FUNCTION_BLOCK PUBLIC Stack_TestSuite EXTENDS TcUnit.FB_TestSuite

// check datatypes are handled correctly
CheckListWorksWithIntegers();
CheckListWorksWithStrings();
CheckListWorksWithArrays();

// all other checks
CheckStackImplementsI_Stack();
CheckContains();
CheckClear();
CheckCount();
CheckAddItem();
CheckTryRemoveItem();
CheckTryPopRemovesTheItem();
CheckTryPopReturnsTheCorrectValue();
CheckTryPeekReturnsTheCorrectValue();
CheckTryPeekDoesNotRemoveTheItem();
CheckOnChangedEvent();
CheckOnDisposedEvent();
CheckOnceEvent();
CheckOffEvent();
CheckTryCopyTo();
CheckTryCopyToLocation();
CheckStackOrderIsCorrect();
CheckListReturnsEnumerator();
CheckEnumeratorIsInvalidAfterChange();
CheckIsEmptyWhenEmpty();
CheckIsEmptyWhenFull();

METHOD PUBLIC CheckAddItem
VAR
	in1 : INT := 123;
	in2 : INT := 456;
	in3 : INT := 789;
	result : BOOL;
	stack : Stack;
END_VAR
TEST('CheckAddItem');

// @TEST-FIXTURE
stack.Push(in1); // (fifo->) 123
stack.Push(in2); // (fifo->) 456, 123

// @TEST-RUN
stack.AddItem(in3); // fifo->) 789, 456, 123
result := stack.Contains(in3);

// @TEST-ASSSERT
AssertTrue(
	Condition := result,
	Message := 'Method returned false'
);

TEST_FINISHED();
END_METHOD

METHOD PUBLIC CheckClear
VAR
	in1 : INT := 123;
	in2 : INT := 456;
	in3 : INT := 789;
	stack : Stack;
END_VAR
TEST('CheckClear');

// @TEST-FIXTURE
stack.Push(in1); // (fifo->) 123
stack.Push(in2); // (fifo->) 456, 123
stack.Push(in2); // (fifo->) 789, 456, 123

// @TEST-RUN
stack.Clear();

// @TEST-ASSSERT
AssertTrue(
	Condition := stack.Count = 0,
	Message := 'The count is not zero'
);

TEST_FINISHED();
END_METHOD

METHOD PUBLIC CheckContains
VAR
	in1 : INT := 123;
	in2 : INT := 456;
	in3 : INT := 789;
	result : BOOL;
	stack : Stack;
END_VAR
TEST('CheckContains');

// @TEST-FIXTURE
stack.Push(in1); // (fifo->) 123
stack.Push(in2); // (fifo->) 456, 123
stack.Push(in2); // (fifo->) 789, 456, 123

// @TEST-RUN
result := stack.Contains(in2);

// @TEST-ASSSERT
AssertTrue(
	Condition := result,
	Message := 'Did not find the item in the queue'
);

TEST_FINISHED();
END_METHOD

METHOD PUBLIC CheckCount
VAR
	in1 : INT := 123;
	in2 : INT := 456;
	in3 : INT := 789;
	total : DINT;
	expected : DINT := 3;
	stack : Stack;
END_VAR
TEST('CheckCount');

// @TEST-FIXTURE
stack.Push(in1); // (fifo->) 123
stack.Push(in2); // (fifo->) 456, 123
stack.Push(in2); // (fifo->) 789, 456, 123

// @TEST-RUN
total := stack.Count;

// @TEST-ASSSERT
AssertEquals(
	Expected := expected,
	Actual := total,
	Message := 'Incorrect count'
);

TEST_FINISHED();
END_METHOD

METHOD PUBLIC CheckEnumeratorIsInvalidAfterChange
VAR
	in : INT := 123;
	result : BOOL;
	stack : Stack;
	enumerator : I_ForwardEnumerator;
END_VAR
TEST('CheckEnumeratorIsInvalidAfterChange');

// @TEST-FIXTURE
enumerator := stack.GetEnumerator();
stack.Push(in);

// @TEST-RUN
result := enumerator.IsValid;
enumerator.Dispose();

// @TEST-ASSSERT
AssertFalse(
	Condition := result,
	Message := 'Method returned true'
);

TEST_FINISHED();
END_METHOD

METHOD PUBLIC CheckIsEmptyWhenEmpty
VAR
	result : BOOL;
	stack : Stack;
END_VAR
TEST('CheckIsEmptyWhenEmpty');

// @TEST-RUN
result := stack.IsEmpty;

// @TEST-ASSSERT
AssertTrue(
	Condition := result,
	Message := 'Incorrect state of IsEmpty'
);

TEST_FINISHED();
END_METHOD

METHOD PUBLIC CheckIsEmptyWhenFull
VAR
	in : INT := 123;
	result : BOOL;
	stack : Stack;
END_VAR
TEST('CheckIsEmptyWhenFull');

// @TEST-FIXTURE
stack.Push(in);

// @TEST-RUN
result := stack.IsEmpty;

// @TEST-ASSSERT
AssertFalse(
	Condition := result,
	Message := 'Incorrect state of IsEmpty'
);

TEST_FINISHED();
END_METHOD

METHOD PUBLIC CheckListReturnsEnumerator
VAR
	in1 : INT := 123;
	in2 : INT := 456;
	in3 : INT := 789;
	enumerator : I_ForwardEnumerator;
	stack : Stack;
END_VAR
TEST('CheckListReturnsEnumerator');

// @TEST-FIXTURE
stack.Push(in1); // (fifo->) 123
stack.Push(in2); // (fifo->) 456, 123
stack.Push(in2); // (fifo->) 789, 456, 123

// @TEST-RUN
enumerator := stack.GetEnumerator();

// @TEST-ASSSERT
AssertTrue(
	Condition := (enumerator <> 0),
	Message := 'Did not return an enumerator'
);

// @TEST-DISPOSE
enumerator.Dispose();

TEST_FINISHED();
END_METHOD

METHOD PUBLIC CheckListWorksWithArrays
VAR
	in : ARRAY [0..1] OF REAL := [0.1,2.3];
	out : ARRAY [0..1] OF REAL;
	expected : ARRAY [0..1] OF REAL := [0.1,2.3];
	result : BOOL;
	stack : Stack;
END_VAR
TEST('CheckListWorksWithArrays');

// @TEST-FIXTURE
stack.Push(in);

// @TEST-RUN
result := stack.TryPop(out);

// @TEST-ASSSERT
AssertTrue(
	Condition := result,
	Message := 'Method returned false'
);

AssertEquals(
	Expected := expected,
	Actual := out,
	Message := 'Did not produce the expected result'
);

TEST_FINISHED();
END_METHOD

METHOD PUBLIC CheckListWorksWithIntegers
VAR
	in : INT := 123;
	out : INT;
	expected : INT := 123;
	result : BOOL;
	stack : Stack;
END_VAR
TEST('CheckListWorksWithIntegers');

// @TEST-FIXTURE
stack.Push(in);

// @TEST-RUN
result := stack.TryPop(out);

// @TEST-ASSSERT
AssertTrue(
	Condition := result,
	Message := 'Method returned false'
);

AssertEquals(
	Expected := expected,
	Actual := out,
	Message := 'Did not produce the expected result'
);

TEST_FINISHED();
END_METHOD

METHOD PUBLIC CheckListWorksWithStrings
VAR
	in : STRING := 'test';
	out : STRING;
	expected : STRING := 'test';
	result : BOOL;
	stack : Stack;
END_VAR
TEST('CheckListWorksWithStrings');

// @TEST-FIXTURE
stack.Push(in);

// @TEST-RUN
result := stack.TryPop(out);

// @TEST-ASSSERT
AssertTrue(
	Condition := result,
	Message := 'Method returned false'
);

AssertEquals(
	Expected := expected,
	Actual := out,
	Message := 'Did not produce the expected result'
);

TEST_FINISHED();
END_METHOD

METHOD PUBLIC CheckOffEvent
VAR
	value : INT := 123;
	stack : Stack;
	handler : CollectionChangedEventHandler(ExpectedOriginator := stack);
END_VAR
TEST('CheckOffEvent');

// @TEST-FIXTURE
stack.OnEvent('OnChanged',handler);
stack.OffEvent('OnChanged',handler);

// @TEST-RUN
stack.Push(value);

// @TEST-ASSSERT
AssertFalse(
	Condition := handler.EventReceived,
	Message := 'OnceEvent emitted the OnChanged event more than once'
);

TEST_FINISHED();
END_METHOD

METHOD PUBLIC CheckOnceEvent
VAR
	value : INT := 123;
	stack : Stack;
	handler : CollectionChangedEventHandler(ExpectedOriginator := stack);
END_VAR
TEST('CheckOnceEvent');

// @TEST-FIXTURE
stack.OnceEvent('OnChanged',handler);
stack.Push(value);
handler.Reset();

// @TEST-RUN
stack.Push(value);

// @TEST-ASSSERT
AssertFalse(
	Condition := handler.EventReceived,
	Message := 'OnceEvent emitted the OnChanged event more than once'
);

TEST_FINISHED();
END_METHOD

METHOD PUBLIC CheckOnChangedEvent
VAR
	value : INT := 123;
	stack : Stack;
	handler : CollectionChangedEventHandler(ExpectedOriginator := stack);
END_VAR
TEST('CheckOnChangedEvent');

// @TEST-FIXTURE
stack.OnEvent('OnChanged',handler);

// @TEST-RUN
stack.Push(value);

// @TEST-ASSSERT
AssertTrue(
	Condition := handler.EventReceived,
	Message := 'Did not emit the OnChanged event'
);

AssertTrue(
	Condition := handler.FromExpectedOriginator,
	Message := 'Did not include itself in the OnChanged event'
);

TEST_FINISHED();
END_METHOD

METHOD PUBLIC CheckOnDisposedEvent
VAR
	value : INT := 123;
	pStack : POINTER TO Stack;
	handler : CollectionDisposedEventHandler(ExpectedOriginator := 0);
END_VAR
TEST('CheckOnDisposedEvent');

// @TEST-FIXTURE
pStack := __NEW(Stack);
handler.SetExpectedOriginator(pStack^);
pStack^.OnEvent('OnDisposed',handler);

// @TEST-RUN
pStack^.Dispose();

// @TEST-ASSSERT
AssertTrue(
	Condition := handler.EventReceived,
	Message := 'Did not emit the OnDisposed event'
);

AssertTrue(
	Condition := handler.FromExpectedOriginator,
	Message := 'Did not include itself in the OnDisposed event'
);

TEST_FINISHED();
END_METHOD

METHOD PUBLIC CheckStackImplementsI_Stack
VAR
	stack : Stack;
    iStack : I_Stack := stack;
    result : BOOL;
END_VAR
TEST('CheckStackImplementsI_Stack');

// @TEST-FIXTURE

// @TEST-RUN
result := iStack <> 0;

// @TEST-ASSSERT
AssertTrue(
	Condition := result,
	Message := 'Did not implement I_Stack'
);

TEST_FINISHED();
END_METHOD

METHOD PUBLIC CheckStackOrderIsCorrect
VAR
	in1 : INT := 123;
	in2 : INT := 456;
	in3 : INT := 789;
	out1, out2, out3 : INT;
	expected1 : INT := 789;
	expected2 : INT := 456;
	expected3 : INT := 123;
	result1, result2, result3 : BOOL;
	stack : Stack;
END_VAR
TEST('CheckStackOrderIsCorrect');

// @TEST-FIXTURE
stack.Push(in1); // (fifo->) 123
stack.Push(in2); // (fifo->) 456, 123
stack.Push(in3); // (fifo->) 789, 456, 123

// @TEST-RUN
result1 := stack.TryPop(out1);
result2 := stack.TryPop(out2);
result3 := stack.TryPop(out3);

// @TEST-ASSSERT
AssertTrue(
	Condition := result1 AND result2 AND result3,
	Message := 'Method returned false'
);

AssertEquals(
	Expected := expected1,
	Actual := out1,
	Message := 'Did not produce the expected result'
);

AssertEquals(
	Expected := expected2,
	Actual := out2,
	Message := 'Did not produce the expected result'
);

AssertEquals(
	Expected := expected3,
	Actual := out3,
	Message := 'Did not produce the expected result'
);

TEST_FINISHED();
END_METHOD

METHOD PUBLIC CheckTryCopyTo
VAR
	in1 : INT := 123;
	in2 : INT := 456;
	in3 : INT := 789;
	out : ARRAY [0..2] OF INT;
	expected : ARRAY [0..2] OF INT := [789,456,123];
	stack : Stack;
END_VAR
TEST('CheckTryCopyTo');

// @TEST-FIXTURE
stack.Push(in1); // (fifo->) 123
stack.Push(in2); // (fifo->) 456, 123
stack.Push(in3); // (fifo->) 789, 456, 123

// @TEST-RUN
stack.TryCopyTo(out);

// @TEST-ASSSERT
AssertEquals(
	Expected := expected,
	Actual := out,
	Message := 'Did not produce the expected result'
);

TEST_FINISHED();
END_METHOD

METHOD PUBLIC CheckTryCopyToLocation
VAR
	in1 : INT := 123;
	in2 : INT := 456;
	in3 : INT := 789;
	out : ARRAY [0..2] OF INT;
	expected : ARRAY [0..2] OF INT := [789,456,123];
	stack : Stack;
END_VAR
TEST('CheckTryCopyToLocation');

// @TEST-FIXTURE
stack.Push(in1); // (fifo->) 123
stack.Push(in2); // (fifo->) 456, 123
stack.Push(in3); // (fifo->) 789, 456, 123

// @TEST-RUN
stack.TryCopyToLocation(ADR(out),SIZEOF(out));

// @TEST-ASSSERT
AssertEquals(
	Expected := expected,
	Actual := out,
	Message := 'Did not produce the expected result'
);

TEST_FINISHED();
END_METHOD

METHOD PUBLIC CheckTryPeekDoesNotRemoveTheItem
VAR
	in : INT := 123;
	out : INT;
	total : DINT;
	expected : DINT := 1;
	stack : Stack;
END_VAR
TEST('CheckTryPeekDoesNotRemoveTheItem');

// @TEST-FIXTURE
stack.Push(in); // (fifo->) 123

// @TEST-RUN
stack.TryPeek(out);
total := stack.Count;

// @TEST-ASSSERT
AssertEquals(
	Expected := expected,
	Actual := total,
	Message := 'Incorrect count'
);

TEST_FINISHED();
END_METHOD

METHOD PUBLIC CheckTryPeekReturnsTheCorrectValue
VAR
	in : INT := 123;
	out : INT;
	expected : INT := 123;
	result : BOOL;
	stack : Stack;
END_VAR
TEST('CheckTryPeekReturnsTheCorrectValue');

// @TEST-FIXTURE
stack.Push(in); // (fifo->) 123

// @TEST-RUN
result := stack.TryPeek(out);

// @TEST-ASSSERT
AssertTrue(
	Condition := result,
	Message := 'Method returned false'
);

AssertEquals(
	Expected := expected,
	Actual := out,
	Message := 'Did not produce the expected result'
);

TEST_FINISHED();
END_METHOD

METHOD PUBLIC CheckTryPopRemovesTheItem
VAR
	in : INT := 123;
	out : INT;
	total : DINT;
	expected : DINT := 0;
	stack : Stack;
END_VAR
TEST('CheckTryPopRemovesTheItem');

// @TEST-FIXTURE
stack.Push(in); // (fifo->) 123

// @TEST-RUN
stack.TryPop(out);
total := stack.Count;

// @TEST-ASSSERT
AssertEquals(
	Expected := expected,
	Actual := total,
	Message := 'Incorrect count'
);

TEST_FINISHED();
END_METHOD

METHOD PUBLIC CheckTryPopReturnsTheCorrectValue
VAR
	in : INT := 123;
	out : INT;
	expected : INT := 123;
	result : BOOL;
	stack : Stack;
END_VAR
TEST('CheckTryDequeueReturnsTheCorrectValue');

// @TEST-FIXTURE
stack.Push(in); // (fifo->) 123

// @TEST-RUN
result := stack.TryPop(out);

// @TEST-ASSSERT
AssertTrue(
	Condition := result,
	Message := 'Method returned false'
);

AssertEquals(
	Expected := expected,
	Actual := out,
	Message := 'Did not produce the expected result'
);

TEST_FINISHED();
END_METHOD

METHOD PUBLIC CheckTryRemoveItem
VAR
	in1 : INT := 123;
	in2 : INT := 456;
	in3 : INT := 789;
	result : BOOL;
	stack : Stack;
END_VAR
TEST('CheckTryRemoveItem');

// @TEST-FIXTURE
stack.Push(in1); // (fifo->) 123
stack.Push(in2); // (fifo->) 456, 123
stack.Push(in3); // (fifo->) 789, 456, 123

// @TEST-RUN
stack.TryRemoveItem(in2); // (lifo->) 789, 123
result := stack.Contains(in2);

// @TEST-ASSSERT
AssertFalse(
	Condition := result,
	Message := 'Method returned true'
);

TEST_FINISHED();
END_METHOD

END_FUNCTION_BLOCK

(* stored: Version 1.1.0.1, ProductVersion 3.1.4024.12
   POU Stack_TestSuite: Id {20dd6e3e-1cc3-43f4-aecb-d08b82736d74}, SpecialFunc None
   Method CheckAddItem: Id {b1407b4b-116a-428f-9dec-c1ea8851de1a}
   Method CheckClear: Id {b0101d26-1872-4bfd-a283-d74e6cd3858e}
   Method CheckContains: Id {0ee28faa-13ca-4639-ba25-962325dddf5b}
   Method CheckCount: Id {bc7bc879-21cf-45b0-a93e-f33a33d1da30}
   Method CheckEnumeratorIsInvalidAfterChange: Id {c46e725b-c2ef-40ed-89ed-a29ed877b5f1}
   Method CheckIsEmptyWhenEmpty: Id {d54d7a9a-efc5-47a5-9564-9078ee5e4b9f}
   Method CheckIsEmptyWhenFull: Id {7ac1d6a7-fba2-44e3-b487-fefc09825c58}
   Method CheckListReturnsEnumerator: Id {039328e2-24d9-41db-9ec3-f971c7e671c5}
   Method CheckListWorksWithArrays: Id {83af885a-a18c-42cb-bd82-f0d76d1607bc}
   Method CheckListWorksWithIntegers: Id {97fd0eb1-152a-4c37-8535-1f0c9b6ad96e}
   Method CheckListWorksWithStrings: Id {ccf32e88-5da2-478a-9695-4c326aa1d0e5}
   Method CheckOffEvent: Id {7e76ba36-d58a-4258-a1a3-1e4adb55809d}
   Method CheckOnceEvent: Id {81289ad1-c5f1-40c5-8d7e-a09c23f59ef5}
   Method CheckOnChangedEvent: Id {1af5bf6d-61b4-43ba-831e-4df7a2d2d7c8}
   Method CheckOnDisposedEvent: Id {ea24f3ac-3f0f-4991-a1be-349effc958b4}
   Method CheckStackImplementsI_Stack: Id {9f17d6e7-99b9-48b8-a1f6-f977c9a72060}
   Method CheckStackOrderIsCorrect: Id {4a59aa65-bb7d-4586-a02b-3fa85c6041bb}
   Method CheckTryCopyTo: Id {9fb697c0-ab92-46cd-a4a2-bcf09ce6d767}
   Method CheckTryCopyToLocation: Id {04778451-d673-4ad2-9578-d96bcc13484c}
   Method CheckTryPeekDoesNotRemoveTheItem: Id {053db073-1601-4d48-9295-6aa12fe00b15}
   Method CheckTryPeekReturnsTheCorrectValue: Id {25897b35-6be7-4f51-bd32-fc4fb9b1f72c}
   Method CheckTryPopRemovesTheItem: Id {3cdfc80c-9761-474c-9852-90031bfc446a}
   Method CheckTryPopReturnsTheCorrectValue: Id {0dabd0b8-5f08-450c-9c2f-0bcd0e95d783}
   Method CheckTryRemoveItem: Id {f25f826b-ad0f-4bf1-8859-5179bf9b1e64} *)
